FUNCTION_BLOCK Preparador_Polimero_HMI (* Service Interface Function Block Type *)
  (* Standard: 61499-2 *)
  (* Version 0.0, 30/03/2026, template *)
  PACKAGE Hidryco.HidrycoLib;
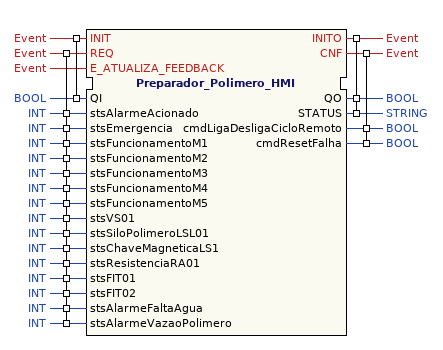
  EVENT_INPUT
    INIT WITH QI;
    REQ WITH stsAlarmeAcionado, stsEmergencia, stsFuncionamentoM1, stsFuncionamentoM2, stsFuncionamentoM3, stsFuncionamentoM4, stsFuncionamentoM5, stsVS01, stsSiloPolimeroLSL01, stsChaveMagneticaLS1, stsResistenciaRA01, stsFIT01, stsFIT02, stsAlarmeFaltaAgua, stsAlarmeVazaoPolimero;
    E_ATUALIZA_FEEDBACK;
  END_EVENT
  EVENT_OUTPUT
    INITO WITH QO, STATUS;
    CNF WITH cmdLigaDesligaCicloRemoto, cmdResetFalha;
  END_EVENT
  VAR_INPUT
    QI : BOOL;
    stsAlarmeAcionado : INT;
    stsEmergencia : INT;
    stsFuncionamentoM1 : INT;
    stsFuncionamentoM2 : INT;
    stsFuncionamentoM3 : INT;
    stsFuncionamentoM4 : INT;
    stsFuncionamentoM5 : INT;
    stsVS01 : INT;
    stsSiloPolimeroLSL01 : INT;
    stsChaveMagneticaLS1 : INT;
    stsResistenciaRA01 : INT;
    stsFIT01 : INT;
    stsFIT02 : INT;
    stsAlarmeFaltaAgua : INT;
    stsAlarmeVazaoPolimero : INT;
  END_VAR
  VAR_OUTPUT
    QO : BOOL; (* Event Output Qualifier *)
    STATUS : STRING; (* Service Status *)
    cmdLigaDesligaCicloRemoto : BOOL;
    cmdResetFalha : BOOL;
  END_VAR
  SERVICE /
    SEQUENCE 
    END_SEQUENCE
  END_SERVICE
END_FUNCTION_BLOCK
